(* IEC 61131-3 sources: CodesysTest/alpha/export/FBs/DataHandlers/FB_ModbusDWORD.pou/HighWord.prop, 1 file *)

(* ---- Get.pm.st ---- *)
(*#-#-#-#-#-#-#-#-#-#---Declaration---#-#-#-#-#-#-#-#-#-#-#-#-#*)

VAR
END_VAR
(*#-#-#-#-#-#-#-#-#-#---Implementation---#-#-#-#-#-#-#-#-#-#-#-#-#*)

HighWord := _highWord;
